// TIA Portal V17 export
// export: Created 2025-06-26T06:49:15.175348Z, ExportSetting WithDefaults, DisplayName Totally Integrated Automation Portal, DisplayVersion V17 Update 8, DisplayName TIA Portal Openness, DisplayVersion V17 Update 8, DisplayName TIA Portal Version Control Interface, DisplayVersion V17, DisplayName STEP 7 Professional, DisplayVersion V17 Update 8, DisplayName STEP 7 Safety, DisplayVersion V17 Update 6, DisplayName WinCC Advanced, DisplayVersion V17 Update 8
FUNCTION_BLOCK "fbHoursCounter"   // FB36, FBD
TITLE = Hours counter
{ S7_Optimized_Access := 'TRUE' }
VERSION : 0.1
// When Enable = TRUE, increase the elapsed time count
// stored: AutoNumber true, IsIECCheckEnabled false, IsRetainMemResEnabled false, MemoryReserve 0, SetENOAutomatically false, UDAEnableTagReadback false
   VAR_INPUT
      bCLK : Bool;   // 1-second pulse
      bEnable : Bool;   // Enable counting
   END_VAR
   VAR_IN_OUT
      sTag : "stHoursCounter";
   END_VAR
   VAR RETAIN
      Hours : CTU_UDINT;
      Minutes { S7_SetPoint := 'True'} : CTU_USINT;
      Seconds { S7_SetPoint := 'True'} : CTU_USINT;
   END_VAR
   VAR
      Rollover_sec { S7_SetPoint := 'True'} : Bool;
      Rollover_min : Bool;
   END_VAR
   VAR_TEMP
      Clock : Bool;
   END_VAR
BEGIN

REGION Network 1: Gate clock bit
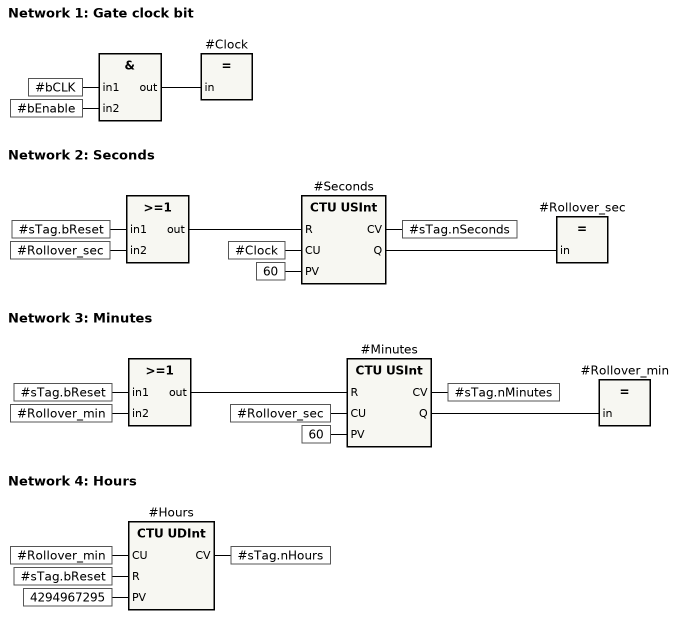
   #Clock := #bCLK AND #bEnable;
END_REGION

REGION Network 2: Seconds
   #Seconds(R := #sTag.bReset OR #Rollover_sec, CU := #Clock, PV := 60, CV => #sTag.nSeconds);   // CTU
   #Rollover_sec := #Seconds.Q;
END_REGION

REGION Network 3: Minutes
   #Minutes(R := #sTag.bReset OR #Rollover_min, CU := #Rollover_sec, PV := 60, CV => #sTag.nMinutes);   // CTU
   #Rollover_min := #Minutes.Q;
END_REGION

REGION Network 4: Hours
   // Note: this is not automatically reset, should count up "forever" (approx equal to 490293 years).
   #Hours(CU := #Rollover_min, R := #sTag.bReset, PV := 4294967295, CV => #sTag.nHours);   // CTU
END_REGION
END_FUNCTION_BLOCK
